FUNCTION_BLOCK DATA_PARSER
  {SET_ATTRIBUTE(OpcUa, SERVICE)}
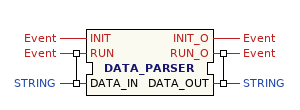
  EVENT_INPUT
    INIT;
    RUN WITH DATA_IN;
  END_EVENT
  EVENT_OUTPUT
    INIT_O;
    RUN_O WITH DATA_OUT;
  END_EVENT
  VAR_INPUT
    DATA_IN : STRING;
  END_VAR
  VAR_OUTPUT
    DATA_OUT : STRING;
  END_VAR
END_FUNCTION_BLOCK
